// TIA Portal V16 export
// export: Created 2022-11-01T21:54:09.3052829Z, ExportSetting WithDefaults, DisplayName Totally Integrated Automation Portal, DisplayVersion V16, DisplayName TIA Portal Version Control Interface, DisplayVersion V16, DisplayName TIA Portal Openness, DisplayVersion V16, DisplayName SINAMICS Startdrive Advanced, DisplayVersion V16, DisplayName SINAMICS Startdrive G130, G150, S120, S150, SINAMICS MV, S210, DisplayVersion V16, DisplayName SINAMICS Startdrive G110M, G120, G120C, G120D, G120P, DisplayVersion V16, DisplayName STEP 7 Professional, DisplayVersion V16, DisplayName STEP 7 Safety, DisplayVersion V16, DisplayName WinCC Professional, DisplayVersion V16
VAR_GLOBAL   // PLC tag table "DI/O C600"
   iH5_Run_Km AT %M10.0 : Bool;   // Работа от сети
   iH5_Con_Vfd AT %M10.1 : Bool;   // Подключен к ТПЧ
   iH5_Run_Vfd AT %M10.2 : Bool;   // Работа ТПЧ
   "qH5_Sel_Loc/Rem" AT %M10.3 : Bool;   // Выбор местный/дистанционный режим
   "qH5_Sel_Km/Vfd" AT %M10.4 : Bool;   // Выбор сеть/ТПЧ
   qH5_Block AT %M10.5 : Bool;   // Блокировка
   qH5_Connect_Vfd AT %M10.6 : Bool;   // Подключить к ТПЧ
   qH5_Start AT %M10.7 : Bool;   // Включить
   iH6_Run_Km AT %M11.0 : Bool;   // Работа от сети
   iH6_Con_Vfd AT %M11.1 : Bool;   // Подключен к ТПЧ
   iH6_Run_Vfd AT %M11.2 : Bool;   // Работа ТПЧ
   "qH6_Sel_Loc/Rem" AT %M11.3 : Bool;   // Выбор местный/дистанционный режим
   "qH6_Sel_Km/Vfd" AT %M11.4 : Bool;   // Выбор сеть/ТПЧ
   qH6_Block AT %M11.5 : Bool;   // Блокировка
   qH6_Connect_Vfd AT %M11.6 : Bool;   // Подключить к ТПЧ
   qH6_Start AT %M11.7 : Bool;   // Включить
   iH13_Run_Km AT %M12.0 : Bool;   // Работа от сети
   iH13_Con_Vfd AT %M12.1 : Bool;   // Подключен к ТПЧ
   iH13_Run_Vfd AT %M12.2 : Bool;   // Работа ТПЧ
   "qH13_Sel_Loc/Rem" AT %M12.3 : Bool;   // Выбор местный/дистанционный режим
   "qH13_Sel_Km/Vfd" AT %M12.4 : Bool;   // Выбор сеть/ТПЧ
   qH13_Block AT %M12.5 : Bool;   // Блокировка
   qH13_Connect_Vfd AT %M12.6 : Bool;   // Подключить к ТПЧ
   qH13_Start AT %M12.7 : Bool;   // Включить
   "iH61/1_Run_Km" AT %M13.0 : Bool;   // Работа от сети
   "iH61/1_Con_Vfd" AT %M13.1 : Bool;   // Подключен к ТПЧ
   "iH61/1_Run_Vfd" AT %M13.2 : Bool;   // Работа ТПЧ
   "qH61/1_Sel_Loc/Rem" AT %M13.3 : Bool;   // Выбор местный/дистанционный режим
   "qH61/1_Sel_Km/Vfd" AT %M13.4 : Bool;   // Выбор сеть/ТПЧ
   "qH61/1_Block" AT %M13.5 : Bool;   // Блокировка
   "qH61/1_Connect_Vfd" AT %M13.6 : Bool;   // Подключить к ТПЧ
   "qH61/1_Start" AT %M13.7 : Bool;   // Включить
   "iH61/2_Run_Km" AT %M14.0 : Bool;   // Работа от сети
   "iH61/2_Con_Vfd" AT %M14.1 : Bool;   // Подключен к ТПЧ
   "iH61/2_Run_Vfd" AT %M14.2 : Bool;   // Работа ТПЧ
   "qH61/2_Sel_Loc/Rem" AT %M14.3 : Bool;   // Выбор местный/дистанционный режим
   "qH61/2_Sel_Km/Vfd" AT %M14.4 : Bool;   // Выбор сеть/ТПЧ
   "qH61/2_Block" AT %M14.5 : Bool;   // Блокировка
   "qH61/2_Connect_Vfd" AT %M14.6 : Bool;   // Подключить к ТПЧ
   "qH61/2_Start" AT %M14.7 : Bool;   // Включить
   "iH62/1_Run_Km" AT %M15.0 : Bool;   // Работа от сети
   "iH62/1_Con_Vfd" AT %M15.1 : Bool;   // Подключен к ТПЧ
   "iH62/1_Run_Vfd" AT %M15.2 : Bool;   // Работа ТПЧ
   "qH62/1_Sel_Loc/Rem" AT %M15.3 : Bool;   // Выбор местный/дистанционный режим
   "qH62/1_Sel_Km/Vfd" AT %M15.4 : Bool;   // Выбор сеть/ТПЧ
   "qH62/1_Block" AT %M15.5 : Bool;   // Блокировка
   "qH62/1_Connect_Vfd" AT %M15.6 : Bool;   // Подключить к ТПЧ
   "qH62/1_Start" AT %M15.7 : Bool;   // Включить
   "iH62/2_Run_Km" AT %M16.0 : Bool;   // Работа от сети
   "iH62/2_Con_Vfd" AT %M16.1 : Bool;   // Подключен к ТПЧ
   "iH62/2_Run_Vfd" AT %M16.2 : Bool;   // Работа ТПЧ
   "qH62/2_Sel_Loc/Rem" AT %M16.3 : Bool;   // Выбор местный/дистанционный режим
   "qH62/2_Sel_Km/Vfd" AT %M16.4 : Bool;   // Выбор сеть/ТПЧ
   "qH62/2_Block" AT %M16.5 : Bool;   // Блокировка
   "qH62/2_Connect_Vfd" AT %M16.6 : Bool;   // Подключить к ТПЧ
   "qH62/2_Start" AT %M16.7 : Bool;   // Включить
   "iH601/1_Run_Km" AT %M17.0 : Bool;   // Работа от сети
   "iH601/1_Con_Vfd" AT %M17.1 : Bool;   // Подключен к ТПЧ
   "iH601/1_Run_Vfd" AT %M17.2 : Bool;   // Работа ТПЧ
   "qH601/1_Sel_Loc/Rem" AT %M17.3 : Bool;   // Выбор местный/дистанционный режим
   "qH601/1_Sel_Km/Vfd" AT %M17.4 : Bool;   // Выбор сеть/ТПЧ
   "qH601/1_Block" AT %M17.5 : Bool;   // Блокировка
   "qH601/1_Connect_Vfd" AT %M17.6 : Bool;   // Подключить к ТПЧ
   "qH601/1_Start" AT %M17.7 : Bool;   // Включить
   "iH601/2_Run_Km" AT %M18.0 : Bool;   // Работа от сети
   "iH601/2_Con_Vfd" AT %M18.1 : Bool;   // Подключен к ТПЧ
   "iH601/2_Run_Vfd" AT %M18.2 : Bool;   // Работа ТПЧ
   "qH601/2_Sel_Loc/Rem" AT %M18.3 : Bool;   // Выбор местный/дистанционный режим
   "qH601/2_Sel_Km/Vfd" AT %M18.4 : Bool;   // Выбор сеть/ТПЧ
   "qH601/2_Block" AT %M18.5 : Bool;   // Блокировка
   "qH601/2_Connect_Vfd" AT %M18.6 : Bool;   // Подключить к ТПЧ
   "qH601/2_Start" AT %M18.7 : Bool;   // Включить
   "iH601/3_Run_Km" AT %M19.0 : Bool;   // Работа от сети
   "iH601/3_Con_Vfd" AT %M19.1 : Bool;   // Подключен к ТПЧ
   "iH601/3_Run_Vfd" AT %M19.2 : Bool;   // Работа ТПЧ
   "qH601/3_Sel_Loc/Rem" AT %M19.3 : Bool;   // Выбор местный/дистанционный режим
   "qH601/3_Sel_Km/Vfd" AT %M19.4 : Bool;   // Выбор сеть/ТПЧ
   "qH601/3_Block" AT %M19.5 : Bool;   // Блокировка
   "qH601/3_Connect_Vfd" AT %M19.6 : Bool;   // Подключить к ТПЧ
   "qH601/3_Start" AT %M19.7 : Bool;   // Включить
   "iH601/4_Run_Km" AT %M20.0 : Bool;   // Работа от сети
   "iH601/4_Con_Vfd" AT %M20.1 : Bool;   // Подключен к ТПЧ
   "iH601/4_Run_Vfd" AT %M20.2 : Bool;   // Работа ТПЧ
   "qH601/4_Sel_Loc/Rem" AT %M20.3 : Bool;   // Выбор местный/дистанционный режим
   "qH601/4_Sel_Km/Vfd" AT %M20.4 : Bool;   // Выбор сеть/ТПЧ
   "qH601/4_Block" AT %M20.5 : Bool;   // Блокировка
   "qH601/4_Connect_Vfd" AT %M20.6 : Bool;   // Подключить к ТПЧ
   "qH601/4_Start" AT %M20.7 : Bool;   // Включить
   "iH601/5_Run_Km" AT %M21.0 : Bool;   // Работа от сети
   "iH601/5_Con_Vfd" AT %M21.1 : Bool;   // Подключен к ТПЧ
   "iH601/5_Run_Vfd" AT %M21.2 : Bool;   // Работа ТПЧ
   "qH601/5_Sel_Loc/Rem" AT %M21.3 : Bool;   // Выбор местный/дистанционный режим
   "qH601/5_Sel_Km/Vfd" AT %M21.4 : Bool;   // Выбор сеть/ТПЧ
   "qH601/5_Block" AT %M21.5 : Bool;   // Блокировка
   "qH601/5_Connect_Vfd" AT %M21.6 : Bool;   // Подключить к ТПЧ
   "qH601/5_Start" AT %M21.7 : Bool;   // Включить
   "iH601/6_Run_Km" AT %M22.0 : Bool;   // Работа от сети
   "iH601/6_Con_Vfd" AT %M22.1 : Bool;   // Подключен к ТПЧ
   "iH601/6_Run_Vfd" AT %M22.2 : Bool;   // Работа ТПЧ
   "qH601/6_Sel_Loc/Rem" AT %M22.3 : Bool;   // Выбор местный/дистанционный режим
   "qH601/6_Sel_Km/Vfd" AT %M22.4 : Bool;   // Выбор сеть/ТПЧ
   "qH601/6_Block" AT %M22.5 : Bool;   // Блокировка
   "qH601/6_Connect_Vfd" AT %M22.6 : Bool;   // Подключить к ТПЧ
   "qH601/6_Start" AT %M22.7 : Bool;   // Включить
   "iH601/7_Run_Km" AT %M23.0 : Bool;   // Работа от сети
   "iH601/7_Con_Vfd" AT %M23.1 : Bool;   // Подключен к ТПЧ
   "iH601/7_Run_Vfd" AT %M23.2 : Bool;   // Работа ТПЧ
   "qH601/7_Sel_Loc/Rem" AT %M23.3 : Bool;   // Выбор местный/дистанционный режим
   "qH601/7_Sel_Km/Vfd" AT %M23.4 : Bool;   // Выбор сеть/ТПЧ
   "qH601/7_Block" AT %M23.5 : Bool;   // Блокировка
   "qH601/7_Connect_Vfd" AT %M23.6 : Bool;   // Подключить к ТПЧ
   "qH601/7_Start" AT %M23.7 : Bool;   // Включить
   "iH602/1_Run_Km" AT %M24.0 : Bool;   // Работа от сети
   "iH602/1_Con_Vfd" AT %M24.1 : Bool;   // Подключен к ТПЧ
   "iH602/1_Run_Vfd" AT %M24.2 : Bool;   // Работа ТПЧ
   "qH602/1_Sel_Loc/Rem" AT %M24.3 : Bool;   // Выбор местный/дистанционный режим
   "qH602/1_Sel_Km/Vfd" AT %M24.4 : Bool;   // Выбор сеть/ТПЧ
   "qH602/1_Block" AT %M24.5 : Bool;   // Блокировка
   "qH602/1_Connect_Vfd" AT %M24.6 : Bool;   // Подключить к ТПЧ
   "qH602/1_Start" AT %M24.7 : Bool;   // Включить
   "iH602/2_Run_Km" AT %M25.0 : Bool;   // Работа от сети
   "iH602/2_Con_Vfd" AT %M25.1 : Bool;   // Подключен к ТПЧ
   "iH602/2_Run_Vfd" AT %M25.2 : Bool;   // Работа ТПЧ
   "qH602/2_Sel_Loc/Rem" AT %M25.3 : Bool;   // Выбор местный/дистанционный режим
   "qH602/2_Sel_Km/Vfd" AT %M25.4 : Bool;   // Выбор сеть/ТПЧ
   "qH602/2_Block" AT %M25.5 : Bool;   // Блокировка
   "qH602/2_Connect_Vfd" AT %M25.6 : Bool;   // Подключить к ТПЧ
   "qH602/2_Start" AT %M25.7 : Bool;   // Включить
   "iH602/3_Run_Km" AT %M26.0 : Bool;   // Работа от сети
   "iH602/3_Con_Vfd" AT %M26.1 : Bool;   // Подключен к ТПЧ
   "iH602/3_Run_Vfd" AT %M26.2 : Bool;   // Работа ТПЧ
   "qH602/3_Sel_Loc/Rem" AT %M26.3 : Bool;   // Выбор местный/дистанционный режим
   "qH602/3_Sel_Km/Vfd" AT %M26.4 : Bool;   // Выбор сеть/ТПЧ
   "qH602/3_Block" AT %M26.5 : Bool;   // Блокировка
   "qH602/3_Connect_Vfd" AT %M26.6 : Bool;   // Подключить к ТПЧ
   "qH602/3_Start" AT %M26.7 : Bool;   // Включить
   "iH602/4_Run_Km" AT %M27.0 : Bool;   // Работа от сети
   "iH602/4_Con_Vfd" AT %M27.1 : Bool;   // Подключен к ТПЧ
   "iH602/4_Run_Vfd" AT %M27.2 : Bool;   // Работа ТПЧ
   "qH602/4_Sel_Loc/Rem" AT %M27.3 : Bool;   // Выбор местный/дистанционный режим
   "qH602/4_Sel_Km/Vfd" AT %M27.4 : Bool;   // Выбор сеть/ТПЧ
   "qH602/4_Block" AT %M27.5 : Bool;   // Блокировка
   "qH602/4_Connect_Vfd" AT %M27.6 : Bool;   // Подключить к ТПЧ
   "qH602/4_Start" AT %M27.7 : Bool;   // Включить
   "iH602/5_Run_Km" AT %M28.0 : Bool;   // Работа от сети
   "iH602/5_Con_Vfd" AT %M28.1 : Bool;   // Подключен к ТПЧ
   "iH602/5_Run_Vfd" AT %M28.2 : Bool;   // Работа ТПЧ
   "qH602/5_Sel_Loc/Rem" AT %M28.3 : Bool;   // Выбор местный/дистанционный режим
   "qH602/5_Sel_Km/Vfd" AT %M28.4 : Bool;   // Выбор сеть/ТПЧ
   "qH602/5_Block" AT %M28.5 : Bool;   // Блокировка
   "qH602/5_Connect_Vfd" AT %M28.6 : Bool;   // Подключить к ТПЧ
   "qH602/5_Start" AT %M28.7 : Bool;   // Включить
   "iH611/1_Run" AT %M29.0 : Bool;   // Работа
   "qH611/1_Start" AT %M29.1 : Bool;   // Включить
   "iH611/2_Run" AT %M29.2 : Bool;   // Работа
   "qH611/2_Start" AT %M29.3 : Bool;   // Включить
   "iH616/1_Run" AT %M29.4 : Bool;   // Работа
   "qH616/1_Start" AT %M29.5 : Bool;   // Включить
   "iH616/2_Run" AT %M29.6 : Bool;   // Работа
   "qH616/2_Start" AT %M29.7 : Bool;   // Включить
   "iBX601/1-1_Run_Vfd" AT %M30.0 : Bool;   // Работа
   "qBX601/1-1_Start" AT %M30.1 : Bool;   // Включить
   "iBX601/1-2_Run_Km" AT %M30.2 : Bool;   // Работа
   "qBX601/1-2_Start" AT %M30.3 : Bool;   // Включить
   "iBX601/1-3_Run_Vfd" AT %M30.4 : Bool;   // Работа
   "qBX601/1-3_Start" AT %M30.5 : Bool;   // Включить
   "iBX601/1-4_Run_Km" AT %M30.6 : Bool;   // Работа
   "qBX601/1-4_Start" AT %M30.7 : Bool;   // Включить
   "iBX601/1-5_Run_Vfd" AT %M31.0 : Bool;   // Работа
   "qBX601/1-5_Start" AT %M31.1 : Bool;   // Включить
   "iBX601/2-1_Run_Vfd" AT %M31.2 : Bool;   // Работа
   "qBX601/2-1_Start" AT %M31.3 : Bool;   // Включить
   "iBX601/2-2_Run_Km" AT %M31.4 : Bool;   // Работа
   "qBX601/2-2_Start" AT %M31.5 : Bool;   // Включить
   "iBX601/2-3_Run_Vfd" AT %M31.6 : Bool;   // Работа
   "qBX601/2-3_Start" AT %M31.7 : Bool;   // Включить
   "iBX601/2-4_Run_Km" AT %M32.0 : Bool;   // Работа
   "qBX601/2-4_Start" AT %M32.1 : Bool;   // Включить
   "iBX601/2-5_Run_Vfd" AT %M32.2 : Bool;   // Работа
   "qBX601/2-5_Start" AT %M32.3 : Bool;   // Включить
   "iBX601/4-1_Run_Km" AT %M32.4 : Bool;   // Работа
   "qBX601/4-1_Start" AT %M32.5 : Bool;   // Включить
   "iBX601/4-2_Run_Km" AT %M32.6 : Bool;   // Работа
   "qBX601/4-2_Start" AT %M32.7 : Bool;   // Включить
   "iBX601/4-3_Run_Km" AT %M33.0 : Bool;   // Работа
   "qBX601/4-3_Start" AT %M33.1 : Bool;   // Включить
   "iBX602/1-1_Run_Vfd" AT %M33.2 : Bool;   // Работа
   "qBX602/1-1_Start" AT %M33.3 : Bool;   // Включить
   "iBX602/1-2_Run_Km" AT %M33.4 : Bool;   // Работа
   "qBX602/1-2_Start" AT %M33.5 : Bool;   // Включить
   "iBX602/1-3_Run_Vfd" AT %M33.6 : Bool;   // Работа
   "qBX602/1-3_Start" AT %M33.7 : Bool;   // Включить
   "iBX602/1-4_Run_Km" AT %M34.0 : Bool;   // Работа
   "qBX602/1-4_Start" AT %M34.1 : Bool;   // Включить
   "iBX602/1-5_Run_Vfd" AT %M34.2 : Bool;   // Работа
   "qBX602/1-5_Start" AT %M34.3 : Bool;   // Включить
   "iBX602/2-1_Run_Vfd" AT %M34.4 : Bool;   // Работа
   "qBX602/2-1_Start" AT %M34.5 : Bool;   // Включить
   "iBX602/2-2_Run_Km" AT %M34.6 : Bool;   // Работа
   "qBX602/2-2_Start" AT %M34.7 : Bool;   // Включить
   "iBX602/2-3_Run_Vfd" AT %M35.0 : Bool;   // Работа
   "qBX602/2-3_Start" AT %M35.1 : Bool;   // Включить
   "iBX602/2-4_Run_Km" AT %M35.2 : Bool;   // Работа
   "qBX602/2-4_Start" AT %M35.3 : Bool;   // Включить
   "iBX602/2-5_Run_Vfd" AT %M35.4 : Bool;   // Работа
   "qBX602/2-5_Start" AT %M35.5 : Bool;   // Включить
   "iBX602/3-1_Run_Vfd" AT %M35.6 : Bool;   // Работа
   "qBX602/3-1_Start" AT %M35.7 : Bool;   // Включить
   "iBX602/3-2_Run_Km" AT %M36.0 : Bool;   // Работа
   "qBX602/3-2_Start" AT %M36.1 : Bool;   // Включить
   "iBX602/3-3_Run_Vfd" AT %M36.2 : Bool;   // Работа
   "qBX602/3-3_Start" AT %M36.3 : Bool;   // Включить
   "iBX602/3-4_Run_Km" AT %M36.4 : Bool;   // Работа
   "qBX602/3-4_Start" AT %M36.5 : Bool;   // Включить
   "iBX602/3-5_Run_Vfd" AT %M36.6 : Bool;   // Работа
   "qBX602/3-5_Start" AT %M36.7 : Bool;   // Включить
   "iBX602/4-1_Run_Km" AT %M37.0 : Bool;   // Работа
   "qBX602/4-1_Start" AT %M37.1 : Bool;   // Включить
   "iBX602/4-2_Run_Km" AT %M37.2 : Bool;   // Работа
   "qBX602/4-2_Start" AT %M37.3 : Bool;   // Включить
   "iBX602/4-3_Run_Km" AT %M37.4 : Bool;   // Работа
   "qBX602/4-3_Start" AT %M37.5 : Bool;   // Включить
   "iBX603/1-1_Run_Vfd" AT %M37.6 : Bool;   // Работа
   "qBX603/1-1_Start" AT %M37.7 : Bool;   // Включить
   "iBX603/1-2_Run_Km" AT %M38.0 : Bool;   // Работа
   "qBX603/1-2_Start" AT %M38.1 : Bool;   // Включить
   "iBX603/1-3_Run_Vfd" AT %M38.2 : Bool;   // Работа
   "qBX603/1-3_Start" AT %M38.3 : Bool;   // Включить
   "iBX603/1-4_Run_Km" AT %M38.4 : Bool;   // Работа
   "qBX603/1-4_Start" AT %M38.5 : Bool;   // Включить
   "iBX603/2-1_Run_Vfd" AT %M38.6 : Bool;   // Работа
   "qBX603/2-1_Start" AT %M38.7 : Bool;   // Включить
   "iBX603/2-2_Run_Km" AT %M39.0 : Bool;   // Работа
   "qBX603/2-2_Start" AT %M39.1 : Bool;   // Включить
   "iBX603/2-3_Run_Vfd" AT %M39.2 : Bool;   // Работа
   "qBX603/2-3_Start" AT %M39.3 : Bool;   // Включить
   "iBX603/2-4_Run_Km" AT %M39.4 : Bool;   // Работа
   "qBX603/2-4_Start" AT %M39.5 : Bool;   // Включить
   iG601_Run_Km AT %M39.6 : Bool;   // Работа
   qG601_Start AT %M39.7 : Bool;   // Включить
   iUV6104_Opn AT %M40.0 : Bool;
   iUV6104_Cls AT %M40.1 : Bool;
   qUV6104 AT %M40.2 : Bool;
   iUV6105_Opn AT %M40.3 : Bool;
   iUV6105_Cls AT %M40.4 : Bool;
   qUV6105 AT %M40.5 : Bool;
   iUV6106_Opn AT %M40.6 : Bool;
   iUV6106_Cls AT %M40.7 : Bool;
   qUV6106 AT %M41.0 : Bool;
   iUV6107_Opn AT %M41.1 : Bool;
   iUV6107_Cls AT %M41.2 : Bool;
   qUV6107 AT %M41.3 : Bool;
   iUV6108_Opn AT %M41.4 : Bool;
   iUV6108_Cls AT %M41.5 : Bool;
   qUV6108 AT %M41.6 : Bool;
   iUV6114_Opn AT %M41.7 : Bool;
   iUV6114_Cls AT %M42.0 : Bool;
   qUV6114 AT %M42.1 : Bool;
   iUV6116_Opn AT %M42.2 : Bool;
   iUV6116_Cls AT %M42.3 : Bool;
   qUV6116 AT %M42.4 : Bool;
   iUV6117_Opn AT %M42.5 : Bool;
   iUV6117_Cls AT %M42.6 : Bool;
   qUV6117 AT %M42.7 : Bool;
   iUV6118_Opn AT %M43.0 : Bool;
   iUV6118_Cls AT %M43.1 : Bool;
   qUV6118 AT %M43.2 : Bool;
   "iH603/1_Run_Km" AT %M43.3 : Bool;   // Работа от сети
   "iH603/1_Con_Vfd" AT %M43.4 : Bool;   // Подключен к ТПЧ
   "iH603/1_Run_Vfd" AT %M43.5 : Bool;   // Работа ТПЧ
   "qH603/1_Sel_Loc/Rem" AT %M43.6 : Bool;   // Выбор местный/дистанционный режим
   "qH603/1_Sel_Km/Vfd" AT %M43.7 : Bool;   // Выбор сеть/ТПЧ
   "qH603/1_Block" AT %M44.0 : Bool;   // Блокировка
   "qH603/1_Connect_Vfd" AT %M44.1 : Bool;   // Подключить к ТПЧ
   "qH603/1_Start" AT %M44.2 : Bool;   // Включить
   "iH603/2_Run_Km" AT %M44.3 : Bool;   // Работа от сети
   "iH603/2_Con_Vfd" AT %M44.4 : Bool;   // Подключен к ТПЧ
   "iH603/2_Run_Vfd" AT %M44.5 : Bool;   // Работа ТПЧ
   "qH603/2_Sel_Loc/Rem" AT %M44.6 : Bool;   // Выбор местный/дистанционный режим
   "qH603/2_Sel_Km/Vfd" AT %M44.7 : Bool;   // Выбор сеть/ТПЧ
   "qH603/2_Block" AT %M45.0 : Bool;   // Блокировка
   "qH603/2_Connect_Vfd" AT %M45.1 : Bool;   // Подключить к ТПЧ
   "qH603/2_Start" AT %M45.2 : Bool;   // Включить
   "iH617/1_Run_Km" AT %M45.3 : Bool;   // Работа от сети
   "iH617/1_Con_Vfd" AT %M45.4 : Bool;   // Подключен к ТПЧ
   "iH617/1_Run_Vfd" AT %M45.5 : Bool;   // Работа ТПЧ
   "qH617/1_Sel_Loc/Rem" AT %M45.6 : Bool;   // Выбор местный/дистанционный режим
   "qH617/1_Sel_Km/Vfd" AT %M45.7 : Bool;   // Выбор сеть/ТПЧ
   "qH617/1_Block" AT %M46.0 : Bool;   // Блокировка
   "qH617/1_Connect_Vfd" AT %M46.1 : Bool;   // Подключить к ТПЧ
   "qH617/1_Start" AT %M46.2 : Bool;   // Включить
   "iH617/2_Run_Km" AT %M46.3 : Bool;   // Работа от сети
   "iH617/2_Con_Vfd" AT %M46.4 : Bool;   // Подключен к ТПЧ
   "iH617/2_Run_Vfd" AT %M46.5 : Bool;   // Работа ТПЧ
   "qH617/2_Sel_Loc/Rem" AT %M46.6 : Bool;   // Выбор местный/дистанционный режим
   "qH617/2_Sel_Km/Vfd" AT %M46.7 : Bool;   // Выбор сеть/ТПЧ
   "qH617/2_Block" AT %M47.0 : Bool;   // Блокировка
   "qH617/2_Connect_Vfd" AT %M47.1 : Bool;   // Подключить к ТПЧ
   "qH617/2_Start" AT %M47.2 : Bool;   // Включить
   iUV6204_Opn AT %M47.3 : Bool;
   iUV6204_Cls AT %M47.4 : Bool;
   qUV6204 AT %M47.5 : Bool;
   iUV6202_Opn AT %M47.6 : Bool;
   iUV6202_Cls AT %M47.7 : Bool;
   qUV6202 AT %M48.0 : Bool;
   iUV6203_Opn AT %M48.1 : Bool;
   iUV6203_Cls AT %M48.2 : Bool;
   qUV6203 AT %M48.3 : Bool;
   iUV6209_Opn AT %M48.4 : Bool;
   iUV6209_Cls AT %M48.5 : Bool;
   qUV6209 AT %M48.6 : Bool;
   iUV6210_Opn AT %M48.7 : Bool;
   iUV6210_Cls AT %M49.0 : Bool;
   qUV6210 AT %M49.1 : Bool;
   iUV6211_Opn AT %M49.2 : Bool;
   iUV6211_Cls AT %M49.3 : Bool;
   qUV6211 AT %M49.4 : Bool;
   iUV6212_Opn AT %M49.5 : Bool;
   iUV6212_Cls AT %M49.6 : Bool;
   qUV6212 AT %M49.7 : Bool;
   "iH612/1_Run_Km" AT %M50.0 : Bool;
   "iH612/1_Con_Vfd" AT %M50.1 : Bool;
   "iH612/1_Run_Vfd" AT %M50.2 : Bool;
   "qH612/1_Sel_Loc/Rem" AT %M50.3 : Bool;
   "qH612/1_Sel_Km/Vfd" AT %M50.4 : Bool;
   "qH612/1_Block" AT %M50.5 : Bool;
   "qH612/1_Connect_Vfd" AT %M50.6 : Bool;
   "qH612/1_Start" AT %M50.7 : Bool;
   "iH612/2_Run_Km" AT %M51.0 : Bool;
   "iH612/2_Con_Vfd" AT %M51.1 : Bool;
   "iH612/2_Run_Vfd" AT %M51.2 : Bool;
   "qH612/2_Sel_Loc/Rem" AT %M51.3 : Bool;
   "qH612/2_Sel_Km/Vfd" AT %M51.4 : Bool;
   "qH612/2_Block" AT %M51.5 : Bool;
   "qH612/2_Connect_Vfd" AT %M51.6 : Bool;
   "qH612/2_Start" AT %M51.7 : Bool;
   "iH613/1_Run_Km" AT %M52.0 : Bool;
   "iH613/1_Con_Vfd" AT %M52.1 : Bool;
   "iH613/1_Run_Vfd" AT %M52.2 : Bool;
   "qH613/1_Sel_Loc/Rem" AT %M52.3 : Bool;
   "qH613/1_Sel_Km/Vfd" AT %M52.4 : Bool;
   "qH613/1_Block" AT %M52.5 : Bool;
   "qH613/1_Connect_Vfd" AT %M52.6 : Bool;
   "qH613/1_Start" AT %M52.7 : Bool;
   "iH613/2_Run_Km" AT %M53.0 : Bool;
   "iH613/2_Con_Vfd" AT %M53.1 : Bool;
   "iH613/2_Run_Vfd" AT %M53.2 : Bool;
   "qH613/2_Sel_Loc/Rem" AT %M53.3 : Bool;
   "qH613/2_Sel_Km/Vfd" AT %M53.4 : Bool;
   "qH613/2_Block" AT %M53.5 : Bool;
   "qH613/2_Connect_Vfd" AT %M53.6 : Bool;
   "qH613/2_Start" AT %M53.7 : Bool;
   "iH614/1_Run_Km" AT %M54.0 : Bool;
   "iH614/1_Con_Vfd" AT %M54.1 : Bool;
   "iH614/1_Run_Vfd" AT %M54.2 : Bool;
   "qH614/1_Sel_Loc/Rem" AT %M54.3 : Bool;
   "qH614/1_Sel_Km/Vfd" AT %M54.4 : Bool;
   "qH614/1_Block" AT %M54.5 : Bool;
   "qH614/1_Connect_Vfd" AT %M54.6 : Bool;
   "qH614/1_Start" AT %M54.7 : Bool;
   "iH614/2_Run_Km" AT %M55.0 : Bool;
   "iH614/2_Con_Vfd" AT %M55.1 : Bool;
   "iH614/2_Run_Vfd" AT %M55.2 : Bool;
   "qH614/2_Sel_Loc/Rem" AT %M55.3 : Bool;
   "qH614/2_Sel_Km/Vfd" AT %M55.4 : Bool;
   "qH614/2_Block" AT %M55.5 : Bool;
   "qH614/2_Connect_Vfd" AT %M55.6 : Bool;
   "qH614/2_Start" AT %M55.7 : Bool;
   "iH614/3_Run_Km" AT %M56.0 : Bool;
   "iH614/3_Con_Vfd" AT %M56.1 : Bool;
   "iH614/3_Run_Vfd" AT %M56.2 : Bool;
   "qH614/3_Sel_Loc/Rem" AT %M56.3 : Bool;
   "qH614/3_Sel_Km/Vfd" AT %M56.4 : Bool;
   "qH614/3_Block" AT %M56.5 : Bool;
   "qH614/3_Connect_Vfd" AT %M56.6 : Bool;
   "qH614/3_Start" AT %M56.7 : Bool;
   "iH614/4_Run_Km" AT %M57.0 : Bool;
   "iH614/4_Con_Vfd" AT %M57.1 : Bool;
   "iH614/4_Run_Vfd" AT %M57.2 : Bool;
   "qH614/4_Sel_Loc/Rem" AT %M57.3 : Bool;
   "qH614/4_Sel_Km/Vfd" AT %M57.4 : Bool;
   "qH614/4_Block" AT %M57.5 : Bool;
   "qH614/4_Connect_Vfd" AT %M57.6 : Bool;
   "qH614/4_Start" AT %M57.7 : Bool;
   iUV6206_Opn AT %M58.0 : Bool;
   iUV6206_Cls AT %M58.1 : Bool;
   qUV6206 AT %M58.2 : Bool;
   iUV6207_Opn AT %M58.6 : Bool;
   iUV6207_Cls AT %M58.7 : Bool;
   qUV6207 AT %M59.0 : Bool;
   iUV6208_Opn AT %M59.1 : Bool;
   iUV6208_Cls AT %M59.2 : Bool;
   qUV6208 AT %M59.3 : Bool;
   iUV6213_Opn AT %M59.4 : Bool;
   iUV6213_Cls AT %M59.5 : Bool;
   qUV6213 AT %M59.6 : Bool;
   iUV6214_Opn AT %M59.7 : Bool;
   iUV6214_Cls AT %M60.0 : Bool;
   qUV6214 AT %M60.1 : Bool;
   iUV6215_Opn AT %M60.2 : Bool;
   iUV6215_Cls AT %M60.3 : Bool;
   qUV6215 AT %M60.4 : Bool;
   iUV6217_Opn AT %M60.5 : Bool;
   iUV6217_Cls AT %M60.6 : Bool;
   qUV6217 AT %M60.7 : Bool;
   "iH605/1_Run_Km" AT %M61.0 : Bool;
   "iH605/1_Con_Vfd" AT %M61.1 : Bool;
   "iH605/1_Run_Vfd" AT %M61.2 : Bool;
   "qH605/1_Sel_Loc/Rem" AT %M61.3 : Bool;
   "qH605/1_Sel_Km/Vfd" AT %M61.4 : Bool;
   "qH605/1_Block" AT %M61.5 : Bool;
   "qH605/1_Connect_Vfd" AT %M61.6 : Bool;
   "qH605/1_Start" AT %M61.7 : Bool;
   "iH605/2_Run_Km" AT %M62.0 : Bool;
   "iH605/2_Con_Vfd" AT %M62.1 : Bool;
   "iH605/2_Run_Vfd" AT %M62.2 : Bool;
   "qH605/2_Sel_Loc/Rem" AT %M62.3 : Bool;
   "qH605/2_Sel_Km/Vfd" AT %M62.4 : Bool;
   "qH605/2_Block" AT %M62.5 : Bool;
   "qH605/2_Connect_Vfd" AT %M62.6 : Bool;
   "qH605/2_Start" AT %M62.7 : Bool;
   "iH6/3_Run_Km" AT %M63.0 : Bool;
   "iH6/3_Con_Vfd" AT %M63.1 : Bool;
   "iH6/3_Run_Vfd" AT %M63.2 : Bool;
   "qH6/3_Sel_Loc/Rem" AT %M63.3 : Bool;
   "qH6/3_Sel_Km/Vfd" AT %M63.4 : Bool;
   "qH6/3_Block" AT %M63.5 : Bool;
   "qH6/3_Connect_Vfd" AT %M63.6 : Bool;
   "qH6/3_Start" AT %M63.7 : Bool;
   "iH6/4_Run_Km" AT %M64.0 : Bool;
   "iH6/4_Con_Vfd" AT %M64.1 : Bool;
   "iH6/4_Run_Vfd" AT %M64.2 : Bool;
   "qH6/4_Sel_Loc/Rem" AT %M64.3 : Bool;
   "qH6/4_Sel_Km/Vfd" AT %M64.4 : Bool;
   "qH6/4_Block" AT %M64.5 : Bool;
   "qH6/4_Connect_Vfd" AT %M64.6 : Bool;
   "qH6/4_Start" AT %M64.7 : Bool;
   "iH6/5_Run_Km" AT %M65.0 : Bool;
   "iH6/5_Con_Vfd" AT %M65.1 : Bool;
   "iH6/5_Run_Vfd" AT %M65.2 : Bool;
   "qH6/5_Sel_Loc/Rem" AT %M65.3 : Bool;
   "qH6/5_Sel_Km/Vfd" AT %M65.4 : Bool;
   "qH6/5_Block" AT %M65.5 : Bool;
   "qH6/5_Connect_Vfd" AT %M65.6 : Bool;
   "qH6/5_Start" AT %M65.7 : Bool;
END_VAR
